FUNCTION_BLOCK ADP_RLS4 (* Offline identification prototype; see docs/adaptive/4diac-design.md *)
  (* Standard: 61499-2 *)
  (* Version 0.1, 2026-09-26, Guilherme *)
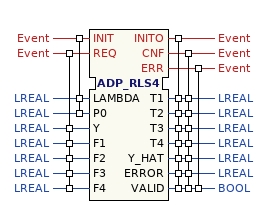
  EVENT_INPUT
    INIT WITH LAMBDA, P0;
    REQ WITH Y, F1, F2, F3, F4;
  END_EVENT
  EVENT_OUTPUT
    INITO WITH T1, T2, T3, T4, Y_HAT, ERROR, VALID;
    CNF WITH T1, T2, T3, T4, Y_HAT, ERROR, VALID;
    ERR WITH VALID;
  END_EVENT
  VAR_INPUT
    LAMBDA : LREAL := 1.0;
    P0 : LREAL := 10000.0;
    Y : LREAL;
    F1 : LREAL;
    F2 : LREAL;
    F3 : LREAL;
    F4 : LREAL;
  END_VAR
  VAR_OUTPUT
    T1 : LREAL;
    T2 : LREAL;
    T3 : LREAL;
    T4 : LREAL;
    Y_HAT : LREAL;
    ERROR : LREAL;
    VALID : BOOL;
  END_VAR
  VAR
    LAMBDA_ACTIVE : LREAL;
    DEN : LREAL;
    V1 : LREAL;
    V2 : LREAL;
    V3 : LREAL;
    V4 : LREAL;
    R1 : LREAL;
    R2 : LREAL;
    R3 : LREAL;
    R4 : LREAL;
    G1 : LREAL;
    G2 : LREAL;
    G3 : LREAL;
    G4 : LREAL;
    N1 : LREAL;
    N2 : LREAL;
    N3 : LREAL;
    N4 : LREAL;
    P11 : LREAL;
    P12 : LREAL;
    P13 : LREAL;
    P14 : LREAL;
    P21 : LREAL;
    P22 : LREAL;
    P23 : LREAL;
    P24 : LREAL;
    P31 : LREAL;
    P32 : LREAL;
    P33 : LREAL;
    P34 : LREAL;
    P41 : LREAL;
    P42 : LREAL;
    P43 : LREAL;
    P44 : LREAL;
    C11 : LREAL;
    C12 : LREAL;
    C13 : LREAL;
    C14 : LREAL;
    C21 : LREAL;
    C22 : LREAL;
    C23 : LREAL;
    C24 : LREAL;
    C31 : LREAL;
    C32 : LREAL;
    C33 : LREAL;
    C34 : LREAL;
    C41 : LREAL;
    C42 : LREAL;
    C43 : LREAL;
    C44 : LREAL;
  END_VAR
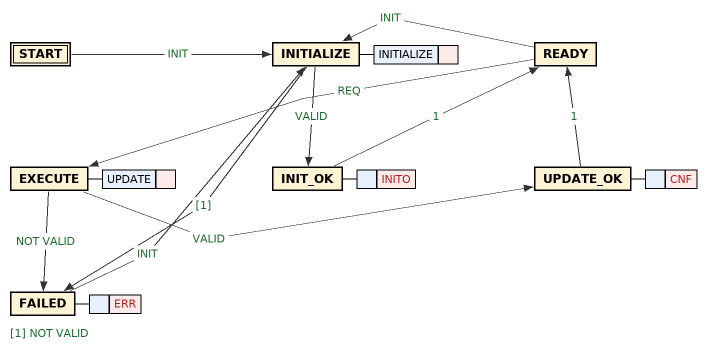
  EC_STATES
    START;
    INITIALIZE : INITIALIZE;
    READY;
    EXECUTE : UPDATE;
    INIT_OK : -> INITO;
    UPDATE_OK : -> CNF;
    FAILED : -> ERR;
  END_STATES
  EC_TRANSITIONS
    START TO INITIALIZE := INIT;
    INITIALIZE TO INIT_OK := VALID;
    INITIALIZE TO FAILED := NOT VALID;
    INIT_OK TO READY := 1;
    READY TO INITIALIZE := INIT;
    READY TO EXECUTE := REQ;
    EXECUTE TO UPDATE_OK := VALID;
    EXECUTE TO FAILED := NOT VALID;
    UPDATE_OK TO READY := 1;
    FAILED TO INITIALIZE := INIT;
  END_TRANSITIONS
  ALGORITHM INITIALIZE IN ST:
VALID := FALSE;
Y_HAT := 0.0;
ERROR := 0.0;
LAMBDA_ACTIVE := LAMBDA;
T1 := 0.0;
T2 := 0.0;
T3 := 0.0;
T4 := 0.0;
P11 := 0.0;
P12 := 0.0;
P13 := 0.0;
P14 := 0.0;
P21 := 0.0;
P22 := 0.0;
P23 := 0.0;
P24 := 0.0;
P31 := 0.0;
P32 := 0.0;
P33 := 0.0;
P34 := 0.0;
P41 := 0.0;
P42 := 0.0;
P43 := 0.0;
P44 := 0.0;
IF (LAMBDA > 0.0) AND (LAMBDA <= 1.0) AND (P0 > 0.0) AND (P0 <= 1.0E100) THEN
P11 := P0;
P22 := P0;
P33 := P0;
P44 := P0;
VALID := TRUE;
END_IF;
  END_ALGORITHM
  ALGORITHM UPDATE IN ST:
VALID := FALSE;
IF (Y >= -1.0E100) AND (Y <= 1.0E100) AND (F1 >= -1.0E100) AND (F1 <= 1.0E100) AND (F2 >= -1.0E100) AND (F2 <= 1.0E100) AND (F3 >= -1.0E100) AND (F3 <= 1.0E100) AND (F4 >= -1.0E100) AND (F4 <= 1.0E100) THEN
Y_HAT := F1 * T1 + F2 * T2 + F3 * T3 + F4 * T4;
ERROR := Y - Y_HAT;
V1 := P11 * F1 + P12 * F2 + P13 * F3 + P14 * F4;
V2 := P21 * F1 + P22 * F2 + P23 * F3 + P24 * F4;
V3 := P31 * F1 + P32 * F2 + P33 * F3 + P34 * F4;
V4 := P41 * F1 + P42 * F2 + P43 * F3 + P44 * F4;
R1 := F1 * P11 + F2 * P21 + F3 * P31 + F4 * P41;
R2 := F1 * P12 + F2 * P22 + F3 * P32 + F4 * P42;
R3 := F1 * P13 + F2 * P23 + F3 * P33 + F4 * P43;
R4 := F1 * P14 + F2 * P24 + F3 * P34 + F4 * P44;
DEN := LAMBDA_ACTIVE + F1 * V1 + F2 * V2 + F3 * V3 + F4 * V4;
IF (DEN > 1.0E-100) AND (DEN <= 1.0E100) THEN
G1 := V1 / DEN;
G2 := V2 / DEN;
G3 := V3 / DEN;
G4 := V4 / DEN;
N1 := T1 + G1 * ERROR;
N2 := T2 + G2 * ERROR;
N3 := T3 + G3 * ERROR;
N4 := T4 + G4 * ERROR;
C11 := (P11 - G1 * R1) / LAMBDA_ACTIVE;
C12 := (P12 - G1 * R2) / LAMBDA_ACTIVE;
C13 := (P13 - G1 * R3) / LAMBDA_ACTIVE;
C14 := (P14 - G1 * R4) / LAMBDA_ACTIVE;
C21 := (P21 - G2 * R1) / LAMBDA_ACTIVE;
C22 := (P22 - G2 * R2) / LAMBDA_ACTIVE;
C23 := (P23 - G2 * R3) / LAMBDA_ACTIVE;
C24 := (P24 - G2 * R4) / LAMBDA_ACTIVE;
C31 := (P31 - G3 * R1) / LAMBDA_ACTIVE;
C32 := (P32 - G3 * R2) / LAMBDA_ACTIVE;
C33 := (P33 - G3 * R3) / LAMBDA_ACTIVE;
C34 := (P34 - G3 * R4) / LAMBDA_ACTIVE;
C41 := (P41 - G4 * R1) / LAMBDA_ACTIVE;
C42 := (P42 - G4 * R2) / LAMBDA_ACTIVE;
C43 := (P43 - G4 * R3) / LAMBDA_ACTIVE;
C44 := (P44 - G4 * R4) / LAMBDA_ACTIVE;
C12 := (C12 + C21) / 2.0;
C21 := C12;
C13 := (C13 + C31) / 2.0;
C31 := C13;
C14 := (C14 + C41) / 2.0;
C41 := C14;
C23 := (C23 + C32) / 2.0;
C32 := C23;
C24 := (C24 + C42) / 2.0;
C42 := C24;
C34 := (C34 + C43) / 2.0;
C43 := C34;
IF (N1 >= -1.0E100) AND (N1 <= 1.0E100) AND (N2 >= -1.0E100) AND (N2 <= 1.0E100) AND (N3 >= -1.0E100) AND (N3 <= 1.0E100) AND (N4 >= -1.0E100) AND (N4 <= 1.0E100) AND (C11 >= -1.0E100) AND (C11 <= 1.0E100) AND (C12 >= -1.0E100) AND (C12 <= 1.0E100) AND (C13 >= -1.0E100) AND (C13 <= 1.0E100) AND (C14 >= -1.0E100) AND (C14 <= 1.0E100) AND (C21 >= -1.0E100) AND (C21 <= 1.0E100) AND (C22 >= -1.0E100) AND (C22 <= 1.0E100) AND (C23 >= -1.0E100) AND (C23 <= 1.0E100) AND (C24 >= -1.0E100) AND (C24 <= 1.0E100) AND (C31 >= -1.0E100) AND (C31 <= 1.0E100) AND (C32 >= -1.0E100) AND (C32 <= 1.0E100) AND (C33 >= -1.0E100) AND (C33 <= 1.0E100) AND (C34 >= -1.0E100) AND (C34 <= 1.0E100) AND (C41 >= -1.0E100) AND (C41 <= 1.0E100) AND (C42 >= -1.0E100) AND (C42 <= 1.0E100) AND (C43 >= -1.0E100) AND (C43 <= 1.0E100) AND (C44 >= -1.0E100) AND (C44 <= 1.0E100) THEN
T1 := N1;
T2 := N2;
T3 := N3;
T4 := N4;
P11 := C11;
P12 := C12;
P13 := C13;
P14 := C14;
P21 := C21;
P22 := C22;
P23 := C23;
P24 := C24;
P31 := C31;
P32 := C32;
P33 := C33;
P34 := C34;
P41 := C41;
P42 := C42;
P43 := C43;
P44 := C44;
VALID := TRUE;
END_IF;
END_IF;
END_IF;
  END_ALGORITHM
END_FUNCTION_BLOCK
